(* PLC project liner_cyclic.project, CODESYS CODESYS V3.5 SP17 Patch 3 *)
(* stored: creationDateTime 1970-01-01T00:00:00, modificationDateTime 1970-01-01T00:00:00 *)

PROGRAM Sensors
  VAR
    LIN_TRAFO : LIN_TRAFO;
    fbFtMinMax : OSCAT_BASIC.FT_MIN_MAX;  (* //////////fbFtMinMax///////////////////////////// *)
    fbFtMinMax2 : OSCAT_BASIC.FT_MIN_MAX;
    bbtn_reset_FtMinMax : BOOL;
    rMin_FtMinMax : REAL;
    rMax_FtMinMax : REAL;
    out_FORCE : REAL;  (* В Н(Ньютонах) *)
    out_FORCE_in_H : REAL;
    blink : blink;
    rMax_out_FORCE_in_H : REAL;
    rMin_out_FORCE_in_H : REAL;
  END_VAR

            ///////////////////////////////////////////////////////////////////////////////	
	//Выставляем датчик силы в ноль
	LIN_TRAFO(
	IN:= GVL.PAI_F1_FORCE_A5, 
	IN_MIN:= rMin_FtMinMax, 
	IN_MAX:= 16383, 
	OUT_MIN:= 0, 
	OUT_MAX:= 5000, 
	OUT=> out_FORCE , 
	ERROR=> );
	
	out_FORCE_in_H := out_FORCE * 10;   //Показания датчика силы в Н(Ньютонах)
	
	//Вычисляем минимальное значение сырых данных с датчика силы
	fbFtMinMax(      
	IN :=  GVL.PAI_F1_FORCE_A5,
	RST := bbtn_reset_FtMinMax,
	mx => rMax_FtMinMax,
	mn => rMin_FtMinMax);
//////////////////////////////////////////////////////////////////////////////////
//Вычисляем экстремумы датчика силы при работе по синусу
	blink(ENABLE := TRUE, TIMELOW := T#1S, TIMEHIGH := T#1S);

	fbFtMinMax2(      
	IN :=  out_FORCE_in_H,
	RST := blink.OUT,
	mx => rMax_out_FORCE_in_H,
	mn => rMin_out_FORCE_in_H);

          
END_PROGRAM
